TYPE ST_Config_Drops :
STRUCT
	stValve: ST_Config_Valve;
	
END_STRUCT
END_TYPE

(* stored: Version 1.1.0.1, ProductVersion 3.1.4019.2
   DUT ST_Config_Drops: Id {98399b7d-8020-4c6a-be77-9180c1755d41} *)
